// TwinCAT 3 PLC project lcls_plc_tst
// ProgramVersion: 3.1.4026.17
// libraries:
//   LCLS Vacuum, * (SLAC - LCLS)
//   Tc2_Standard, * (Beckhoff Automation GmbH)
//   Tc2_System, * (Beckhoff Automation GmbH)
// project tree:
//   GVLs/ GVL.TcGVL
//   / PlcTask.TcTTO
//   POUs/ MAIN.TcPOU
// real-time tasks:
//   TASK PlcTask: cycle T#10ms, priority 20, ADS port 350
// I/O:
//   DEVICE Device 1 (EtherCAT), AmsNetId 172.21.148.160.2.1
//     Term 9 (EK1200) [EK1200-5000 EtherCAT Power supply (2A E-Bus)]
//       Term 10 (EK1122) [EK1122 2 port EtherCAT junction]
//         Term 11 (EK1100) [EK1100 EtherCAT Coupler (2A E-Bus)]
//           Term 12 (EL2794) [EL2794 4Ch. Dig. Output 24V AC/DC, 2A, short-circuit-proof]
//           Term 13 (EL2794) [EL2794 4Ch. Dig. Output 24V AC/DC, 2A, short-circuit-proof]
//           Term 14 (EL1004) [EL1004 4Ch. Dig. Input 24V, 3ms]
//           Term 15 (EL3174-0042) [EL3174-0042 4Ch. Ana. Input +/-30V, +/-60V 16 Bit, Isolated Channels]
//           Term 18 (EL9011)
//         Box 16 (EP2338-0002) [EP2338-0002 8 Ch. Dig. Input/Output 24V, 0,5A, M12]
//         Box 17 (EP2624-0002) [EP2624-0002 4Ch. Relay Output, NO (125V AC / 30V DC)]
// variable links:
//   (this object) <-> Device 1 (EtherCAT)/Term 9 (EK1200)/Term 10 (EK1122)/Box 16 (EP2338-0002)
//     PlcTask Inputs/GVL.test_pump_2.i_xAlarm <-> Channel 1/Input
//     PlcTask Inputs/GVL.test_pump_2.i_xIsRun <-> Channel 2/Input
//   (this object) <-> Device 1 (EtherCAT)/Term 9 (EK1200)/Term 10 (EK1122)/Box 17 (EP2624-0002)
//     PlcTask Outputs/GVL.test_pump_2.q_xLspdDo <-> Channel 3/Output
//     PlcTask Outputs/GVL.test_pump_2.q_xRemote <-> Channel 2/Output
//     PlcTask Outputs/GVL.test_pump_2.q_xResetDo <-> Channel 4/Output
//     PlcTask Outputs/GVL.test_pump_2.q_xRunDO <-> Channel 1/Output

CONFIGURATION lcls_plc_tst
    RESOURCE PLC ON TwinCAT3
        TASK PlcTask(INTERVAL := T#10ms, PRIORITY := 20);
        PROGRAM MAIN WITH PlcTask : MAIN;
    END_RESOURCE
END_CONFIGURATION

// ---- GVLs/GVL.TcGVL
//{attribute 'qualified_only'}
VAR_GLOBAL
	{attribute 'pytmc' := 'pv: TEST:PUMP:KASHIYAMA'}
	{attribute 'TcLinkTo' := 	'.q_xRunDO 			:=	TIIB[Term 5 (EL2794)]^Channel 1^Output;
                                 .q_xRemote		:=	TIIB[Term 5 (EL2794)]^Channel 2^Output;
                                 .q_xLspdDo			:=	TIIB[Term 5 (EL2794)]^Channel 3^Output;
                                 .q_xResetDo 		:=	TIIB[Term 5 (EL2794)]^Channel 4^Output;
                                 .i_xAlarm	:=	TIIB[Term 6 (EL1004)]^Channel 2^Input;
                                 .i_xIsRun	:=	TIIB[Term 6 (EL1004)]^Channel 1^Input
    '}
	test_pump : FB_KashiyamaPump_G;
	
	{attribute 'pytmc' := 'pv: TEST:PUMP:KASHIYAMA:02'}
	{attribute 'TcLinkTo' := 	'.q_xRunDO 			:=	TIIB[Box 17 (EP2624-0002)]^Channel 1^Output;
                                 .q_xRemote		:=	TIIB[Box 17 (EP2624-0002)]^Channel 2^Output;
                                 .q_xLspdDo			:=	TIIB[Box 17 (EP2624-0002)]^Channel 3^Output;
                                 .q_xResetDo 		:=	TIIB[Box 17 (EP2624-0002)]^Channel 4^Output;
                                 .i_xAlarm	:=	TIIB[Box 16 (EP2338-0002)]^Channel 1^Input;
                                 .i_xIsRun	:=	TIIB[Box 16 (EP2338-0002)]^Channel 2^Input
    '}
	test_pump_2 : FB_KashiyamaPump_G;
	
END_VAR

// ---- POUs/MAIN.TcPOU
PROGRAM MAIN
VAR
	{attribute 'pytmc' := 'pv: TEST:NEODRY:01'}
	test : BOOL;
END_VAR

test_pump();

test_pump_2();

END_PROGRAM
